KUKA KRL program: makrosps.src

&ACCESS RVO1
&COMMENT MAKRO_SPS_BASIC
&PARAM TEMPLATE = C:\KRC\Roboter\Template\makrospsvorgabe.src
&PARAM TPVW_VERSION = 8.1.8
&PARAM EDITMASK = MakroSPS
DEF MAKROSPS()
   ;FOLD Makro Anfang ;%{PSE}%MKUKATPVW
      SPS_N=-1
   ;ENDFOLD
   ;FOLD -- Freilaufende  SPS  (Basic) -- ;%{E}%MKUKATPVW %CVW_COM %VCOMMENT %P 2:-- Freilaufende  SPS  (Basic) --, 3: VW_COMMENT
   ;ENDFOLD
   ;FOLD -- KS24 -- ;%{E}%MKUKATPVW %CVW_COM %VCOMMENT %P 2:-- KS24 --, 3: VW_COMMENT
   ;ENDFOLD
   ;FOLD -- Version: 01 -- ;%{E}%MKUKATPVW %CVW_COM %VCOMMENT %P 2:-- Version: 01 --, 3: VW_COMMENT
   ;ENDFOLD
   ;FOLD -- Stand: 008 -- ;%{E}%MKUKATPVW %CVW_COM %VCOMMENT %P 2:-- Stand: 008 --, 3: VW_COMMENT
   ;ENDFOLD
   ;FOLD -- letzte  Aenderung  02.11.2017 LZ -- ;%{E}%MKUKATPVW %CVW_COM %VCOMMENT %P 2:-- letzte  Aenderung  02.11.2017 LZ --, 3: VW_COMMENT
   ;ENDFOLD
   ;FOLD -- Hilfszeit MakroSPS -- ;%{E}%MKUKATPVW %CVW_COM %VCOMMENT %P 2:-- Hilfszeit MakroSPS --, 3: VW_COMMENT
   ;ENDFOLD
   ;FOLD t20 ( !A4060 ) = -35[1/10Sek] ;%{E}%MKUKATPVW %CVW_SPS %VTASG %P 2:t20 ( !A4060 ) = -35[1/10Sek], 3: TASG
      VW(#SET_TIME,NOT $OUT[4060],20,0,-35)
   ;ENDFOLD
   ;FOLD -- Hilfsflags fuer Medien -- ;%{E}%MKUKATPVW %CVW_COM %VCOMMENT %P 2:-- Hilfsflags fuer Medien --, 3: VW_COMMENT
   ;ENDFOLD
   ;FOLD F127 = (!F734 & E514 & E515) + (F734 & E517 & E518) ;%{E}%MKUKATPVW %CVW_SPS %VBOASG %P 2:F127 = (!F734 & E514 & E515) + (F734 & E517 & E518), 3: BOASG
      $FLAG[127] = (NOT $FLAG[734] AND $IN[514] AND $IN[515]) OR ($FLAG[734] AND $IN[517] AND $IN[518])
   ;ENDFOLD
   ;FOLD F162 = E522 & E523 ;%{E}%MKUKATPVW %CVW_SPS %VBOASG %P 2:F162 = E522 & E523, 3: BOASG
      $FLAG[162] = $IN[522] AND $IN[523]
   ;ENDFOLD
   ;FOLD F198 = E530 & E531 ;%{E}%MKUKATPVW %CVW_SPS %VBOASG %P 2:F198 = E530 & E531, 3: BOASG
      $FLAG[198] = $IN[530] AND $IN[531]
   ;ENDFOLD
   ;FOLD -- Reset Motorsteuermodul KF 1 -- ;%{E}%MKUKATPVW %CVW_COM %VCOMMENT %P 2:-- Reset Motorsteuermodul KF 1 --, 3: VW_COMMENT
   ;ENDFOLD
   ;FOLD A833 = !T20 & E840 & A4060 + E840 & E26 ;%{E}%MKUKATPVW %CVW_SPS %VBOASG %P 2:A833 = !T20 & E840 & A4060 + E840 & E26, 3: BOASG
      $OUT[833] = NOT $TIMER_FLAG[20] AND $IN[840] AND $OUT[4060] OR $IN[840] AND $IN[26]
   ;ENDFOLD
   ;FOLD -- Reset Motorsteuermodul KS 1 -- ;%{E}%MKUKATPVW %CVW_COM %VCOMMENT %P 2:-- Reset Motorsteuermodul KS 1 --, 3: VW_COMMENT
   ;ENDFOLD
   ;FOLD A841 = !T20 & E848 & A4060 + E848 & E26 ;%{E}%MKUKATPVW %CVW_SPS %VBOASG %P 2:A841 = !T20 & E848 & A4060 + E848 & E26, 3: BOASG
      $OUT[841] = NOT $TIMER_FLAG[20] AND $IN[848] AND $OUT[4060] OR $IN[848] AND $IN[26]
   ;ENDFOLD
   ;FOLD -- Reset Motorsteuermodul ZS 1 -- ;%{E}%MKUKATPVW %CVW_COM %VCOMMENT %P 2:-- Reset Motorsteuermodul ZS 1 --, 3: VW_COMMENT
   ;ENDFOLD
   ;FOLD A849 = !T20 & E856 & A4060 + E856 & E26 ;%{E}%MKUKATPVW %CVW_SPS %VBOASG %P 2:A849 = !T20 & E856 & A4060 + E856 & E26, 3: BOASG
      $OUT[849] = NOT $TIMER_FLAG[20] AND $IN[856] AND $OUT[4060] OR $IN[856] AND $IN[26]
   ;ENDFOLD
   ;FOLD -- Reset Motorsteuermodul KF 2 -- ;%{E}%MKUKATPVW %CVW_COM %VCOMMENT %P 2:-- Reset Motorsteuermodul KF 2 --, 3: VW_COMMENT
   ;ENDFOLD
   ;FOLD A993 = !T20 & E1000 & A4060 + E1000 & E26 ;%{E}%MKUKATPVW %CVW_SPS %VBOASG %P 2:A993 = !T20 & E1000 & A4060 + E1000 & E26, 3: BOASG
      $OUT[993] = NOT $TIMER_FLAG[20] AND $IN[1000] AND $OUT[4060] OR $IN[1000] AND $IN[26]
   ;ENDFOLD
   ;FOLD -- Reset Motorsteuermodul KS 2 -- ;%{E}%MKUKATPVW %CVW_COM %VCOMMENT %P 2:-- Reset Motorsteuermodul KS 2 --, 3: VW_COMMENT
   ;ENDFOLD
   ;FOLD A1001 = !T20 & E1008 & A4060 + E1008 & E26 ;%{E}%MKUKATPVW %CVW_SPS %VBOASG %P 2:A1001 = !T20 & E1008 & A4060 + E1008 & E26, 3: BOASG
      $OUT[1001] = NOT $TIMER_FLAG[20] AND $IN[1008] AND $OUT[4060] OR $IN[1008] AND $IN[26]
   ;ENDFOLD
   ;FOLD -- Reset Motorsteuermodul ZS 2 -- ;%{E}%MKUKATPVW %CVW_COM %VCOMMENT %P 2:-- Reset Motorsteuermodul ZS 2 --, 3: VW_COMMENT
   ;ENDFOLD
   ;FOLD A1009 = !T20 & E1016 & A4060 + E1016 & E26 ;%{E}%MKUKATPVW %CVW_SPS %VBOASG %P 2:A1009 = !T20 & E1016 & A4060 + E1016 & E26, 3: BOASG
      $OUT[1009] = NOT $TIMER_FLAG[20] AND $IN[1016] AND $OUT[4060] OR $IN[1016] AND $IN[26]
   ;ENDFOLD
   ;FOLD -- Reset Motorsteuermodul KF 3 -- ;%{E}%MKUKATPVW %CVW_COM %VCOMMENT %P 2:-- Reset Motorsteuermodul KF 3 --, 3: VW_COMMENT
   ;ENDFOLD
   ;FOLD A1153 = !T20 & E1160 & A4060 + E1160 & E26 ;%{E}%MKUKATPVW %CVW_SPS %VBOASG %P 2:A1153 = !T20 & E1160 & A4060 + E1160 & E26, 3: BOASG
      $OUT[1153] = NOT $TIMER_FLAG[20] AND $IN[1160] AND $OUT[4060] OR $IN[1160] AND $IN[26]
   ;ENDFOLD
   ;FOLD -- Reset Motorsteuermodul KS 3 -- ;%{E}%MKUKATPVW %CVW_COM %VCOMMENT %P 2:-- Reset Motorsteuermodul KS 3 --, 3: VW_COMMENT
   ;ENDFOLD
   ;FOLD A1161 = !T20 & E1168 & A4060 + E1168 & E26 ;%{E}%MKUKATPVW %CVW_SPS %VBOASG %P 2:A1161 = !T20 & E1168 & A4060 + E1168 & E26, 3: BOASG
      $OUT[1161] = NOT $TIMER_FLAG[20] AND $IN[1168] AND $OUT[4060] OR $IN[1168] AND $IN[26]
   ;ENDFOLD
   ;FOLD -- Reset Motorsteuermodul ZS 2 -- ;%{E}%MKUKATPVW %CVW_COM %VCOMMENT %P 2:-- Reset Motorsteuermodul ZS 2 --, 3: VW_COMMENT
   ;ENDFOLD
   ;FOLD A1169 = !T20 & E1176 & A4060 + E1176 & E26 ;%{E}%MKUKATPVW %CVW_SPS %VBOASG %P 2:A1169 = !T20 & E1176 & A4060 + E1176 & E26, 3: BOASG
      $OUT[1169] = NOT $TIMER_FLAG[20] AND $IN[1176] AND $OUT[4060] OR $IN[1176] AND $IN[26]
   ;ENDFOLD
   ;FOLD -- FK von SK1 abspeichern -- ;%{E}%MKUKATPVW %CVW_COM %VCOMMENT %P 2:-- FK von SK1 abspeichern --, 3: VW_COMMENT
   ;ENDFOLD
   ;FOLD F80 = E804 & !E806 & !E775 & E785 + E785 & E15 + F80 & A785 + F525 + E145 ;%{E}%MKUKATPVW %CVW_SPS %VBOASG %P 2:F80 = E804 & !E806 & !E775 & E785 + E785 & E15 + F80 & A785 + F525 + E145, 3: BOASG
      $FLAG[80] = $IN[804] AND NOT $IN[806] AND NOT $IN[775] AND $IN[785] OR $IN[785] AND $IN[15] OR $FLAG[80] AND $OUT[785] OR $FLAG[525] OR $IN[145]
   ;ENDFOLD
   ;FOLD -- FK von Kombi 1 abspeichern -- ;%{E}%MKUKATPVW %CVW_COM %VCOMMENT %P 2:-- FK von Kombi 1 abspeichern --, 3: VW_COMMENT
   ;ENDFOLD
   ;FOLD F833 = E787 & !E789 & !E775 & E719 + E719 & E15 + F833 & A718 + F525 + E130 ;%{E}%MKUKATPVW %CVW_SPS %VBOASG %P 2:F833 = E787 & !E789 & !E775 & E719 + E719 & E15 + F833 & A718 + F525 + E130, 3: BOASG
      $FLAG[833] = $IN[787] AND NOT $IN[789] AND NOT $IN[775] AND $IN[719] OR $IN[719] AND $IN[15] OR $FLAG[833] AND $OUT[718] OR $FLAG[525] OR $IN[130]
   ;ENDFOLD
   ;FOLD -- FK von SK2 abspeichern -- ;%{E}%MKUKATPVW %CVW_COM %VCOMMENT %P 2:-- FK von SK2 abspeichern --, 3: VW_COMMENT
   ;ENDFOLD
   ;FOLD F140 = E964 & !E966 & !E935 & E945 + E945 & E15 + F140 & A945 + F525 + E177 ;%{E}%MKUKATPVW %CVW_SPS %VBOASG %P 2:F140 = E964 & !E966 & !E935 & E945 + E945 & E15 + F140 & A945 + F525 + E177, 3: BOASG
      $FLAG[140] = $IN[964] AND NOT $IN[966] AND NOT $IN[935] AND $IN[945] OR $IN[945] AND $IN[15] OR $FLAG[140] AND $OUT[945] OR $FLAG[525] OR $IN[177]
   ;ENDFOLD
   ;FOLD -- FK von Kombi 2 abspeichern -- ;%{E}%MKUKATPVW %CVW_COM %VCOMMENT %P 2:-- FK von Kombi 2 abspeichern --, 3: VW_COMMENT
   ;ENDFOLD
   ;FOLD F834 = E947 & !E949 & !E935 & E879 + E879 & E15 + F834 & A878 + F525 + E162 ;%{E}%MKUKATPVW %CVW_SPS %VBOASG %P 2:F834 = E947 & !E949 & !E935 & E879 + E879 & E15 + F834 & A878 + F525 + E162, 3: BOASG
      $FLAG[834] = $IN[947] AND NOT $IN[949] AND NOT $IN[935] AND $IN[879] OR $IN[879] AND $IN[15] OR $FLAG[834] AND $OUT[878] OR $FLAG[525] OR $IN[162]
   ;ENDFOLD
   ;FOLD -- FK von SK3 abspeichern -- ;%{E}%MKUKATPVW %CVW_COM %VCOMMENT %P 2:-- FK von SK3 abspeichern --, 3: VW_COMMENT
   ;ENDFOLD
   ;FOLD F176 = E1124 & !E1126 & !E1095 & E1105 + E1105 & E15 + F176 & A1105 + F525 + E209 ;%{E}%MKUKATPVW %CVW_SPS %VBOASG %P 2:F176 = E1124 & !E1126 & !E1095 & E1105 + E1105 & E15 + F176 & A1105 + F525 + E209, 3: BOASG
      $FLAG[176] = $IN[1124] AND NOT $IN[1126] AND NOT $IN[1095] AND $IN[1105] OR $IN[1105] AND $IN[15] OR $FLAG[176] AND $OUT[1105] OR $FLAG[525] OR $IN[209]
   ;ENDFOLD
   ;FOLD -- FK von Kombi 3 abspeichern -- ;%{E}%MKUKATPVW %CVW_COM %VCOMMENT %P 2:-- FK von Kombi 3 abspeichern --, 3: VW_COMMENT
   ;ENDFOLD
   ;FOLD F835 = E1107 & !E1109 & !E1095 & E1039 + E1039 & E15 + F835 & A1038 + F525 + E194 ;%{E}%MKUKATPVW %CVW_SPS %VBOASG %P 2:F835 = E1107 & !E1109 & !E1095 & E1039 + E1039 & E15 + F835 & A1038 + F525 + E194, 3: BOASG
      $FLAG[835] = $IN[1107] AND NOT $IN[1109] AND NOT $IN[1095] AND $IN[1039] OR $IN[1039] AND $IN[15] OR $FLAG[835] AND $OUT[1038] OR $FLAG[525] OR $IN[194]
   ;ENDFOLD
   ;FOLD -- BZ1 -- ;%{E}%MKUKATPVW %CVW_COM %VCOMMENT %P 2:-- BZ1 --, 3: VW_COMMENT
   ;ENDFOLD
   ;FOLD -- A1702 = (!E1697 + !E1699) & E26 -- ;%{E}%MKUKATPVW %CVW_COM %VCOMMENT %P 2:-- A1702 = (!E1697 + !E1699) & E26 --, 3: VW_COMMENT
   ;ENDFOLD
   ;FOLD -- BZ2 -- ;%{E}%MKUKATPVW %CVW_COM %VCOMMENT %P 2:-- BZ2 --, 3: VW_COMMENT
   ;ENDFOLD
   ;FOLD -- A1750 = (!E1745 + !E1747) & E26 -- ;%{E}%MKUKATPVW %CVW_COM %VCOMMENT %P 2:-- A1750 = (!E1745 + !E1747) & E26 --, 3: VW_COMMENT
   ;ENDFOLD
   ;FOLD -- MS1 -- ;%{E}%MKUKATPVW %CVW_COM %VCOMMENT %P 2:-- MS1 --, 3: VW_COMMENT
   ;ENDFOLD
   ;FOLD A1857 = EIN ;%{E}%MKUKATPVW %CVW_SPS %VBOASG %P 2:A1857 = EIN, 3: BOASG
      $OUT[1857] = TRUE
   ;ENDFOLD
   ;FOLD A1858 = !E1858 & (E26 + E27 + !T20 & A4060) ;%{E}%MKUKATPVW %CVW_SPS %VBOASG %P 2:A1858 = !E1858 & (E26 + E27 + !T20 & A4060), 3: BOASG
      $OUT[1858] = NOT $IN[1858] AND ($IN[26] OR $IN[27] OR NOT $TIMER_FLAG[20] AND $OUT[4060])
   ;ENDFOLD
   ;FOLD F570 = A9 & A16 & A4060 & A4039 & E1857 & E1874 & (F960 + F597 & !E128) ;%{E}%MKUKATPVW %CVW_SPS %VBOASG %P 2:F570 = A9 & A16 & A4060 & A4039 & E1857 & E1874 & (F960 + F597 & !E128), 3: BOASG
      $FLAG[570] = $OUT[9] AND $OUT[16] AND $OUT[4060] AND $OUT[4039] AND $IN[1857] AND $IN[1874] AND ($FLAG[960] OR $FLAG[597] AND NOT $IN[128])
   ;ENDFOLD
   ;FOLD A1859 = A12 & E12 & F570 & F571 & (E1859 + !E26) + E211 & F570 & F571 ;%{E}%MKUKATPVW %CVW_SPS %VBOASG %P 2:A1859 = A12 & E12 & F570 & F571 & (E1859 + !E26) + E211 & F570 & F571, 3: BOASG
      $OUT[1859] = $OUT[12] AND $IN[12] AND $FLAG[570] AND $FLAG[571] AND ($IN[1859] OR NOT $IN[26]) OR $IN[211] AND $FLAG[570] AND $FLAG[571]
   ;ENDFOLD
   ;FOLD -- MS2 -- ;%{E}%MKUKATPVW %CVW_COM %VCOMMENT %P 2:-- MS2 --, 3: VW_COMMENT
   ;ENDFOLD
   ;FOLD A1889 = EIN ;%{E}%MKUKATPVW %CVW_SPS %VBOASG %P 2:A1889 = EIN, 3: BOASG
      $OUT[1889] = TRUE
   ;ENDFOLD
   ;FOLD A1890 = !E1890 & (E26 + E27 + !T20 & A4060) ;%{E}%MKUKATPVW %CVW_SPS %VBOASG %P 2:A1890 = !E1890 & (E26 + E27 + !T20 & A4060), 3: BOASG
      $OUT[1890] = NOT $IN[1890] AND ($IN[26] OR $IN[27] OR NOT $TIMER_FLAG[20] AND $OUT[4060])
   ;ENDFOLD
   ;FOLD F579 = A9 & A16 & A4060 & A4039 & E1889 & E1906 & (F960 + F597 & !E128) ;%{E}%MKUKATPVW %CVW_SPS %VBOASG %P 2:F579 = A9 & A16 & A4060 & A4039 & E1889 & E1906 & (F960 + F597 & !E128), 3: BOASG
      $FLAG[579] = $OUT[9] AND $OUT[16] AND $OUT[4060] AND $OUT[4039] AND $IN[1889] AND $IN[1906] AND ($FLAG[960] OR $FLAG[597] AND NOT $IN[128])
   ;ENDFOLD
   ;FOLD A1891 = A12 & E12 & F579 & F580 & (E1891 + !E26) + E203 & F579 & F580 ;%{E}%MKUKATPVW %CVW_SPS %VBOASG %P 2:A1891 = A12 & E12 & F579 & F580 & (E1891 + !E26) + E203 & F579 & F580, 3: BOASG
      $OUT[1891] = $OUT[12] AND $IN[12] AND $FLAG[579] AND $FLAG[580] AND ($IN[1891] OR NOT $IN[26]) OR $IN[203] AND $FLAG[579] AND $FLAG[580]
   ;ENDFOLD
   ;FOLD -- KL1 -- ;%{E}%MKUKATPVW %CVW_COM %VCOMMENT %P 2:-- KL1 --, 3: VW_COMMENT
   ;ENDFOLD
   ;FOLD A1527 = A10 + E1568 ;%{E}%MKUKATPVW %CVW_SPS %VBOASG %P 2:A1527 = A10 + E1568, 3: BOASG
      $OUT[1527] = $OUT[10] OR $IN[1568]
   ;ENDFOLD
   ;FOLD A1528 = A12 ;%{E}%MKUKATPVW %CVW_SPS %VBOASG %P 2:A1528 = A12, 3: BOASG
      $OUT[1528] = $OUT[12]
   ;ENDFOLD
   ;FOLD F339 = (A1529 + A1535 + E9 & !E15 & !F336) & !E1551 & A10 ;%{E}%MKUKATPVW %CVW_SPS %VBOASG %P 2:F339 = (A1529 + A1535 + E9 & !E15 & !F336) & !E1551 & A10, 3: BOASG
      $FLAG[339] = ($OUT[1529] OR $OUT[1535] OR $IN[9] AND NOT $IN[15] AND NOT $FLAG[336]) AND NOT $IN[1551] AND $OUT[10]
   ;ENDFOLD
   ;FOLD A1547 = (F339 & !T20 + F337 + E168) & F542 ;%{E}%MKUKATPVW %CVW_SPS %VBOASG %P 2:A1547 = (F339 & !T20 + F337 + E168) & F542, 3: BOASG
      $OUT[1547] = ($FLAG[339] AND NOT $TIMER_FLAG[20] OR $FLAG[337] OR $IN[168]) AND $FLAG[542]
   ;ENDFOLD
   ;FOLD A1550 = (F339 & !T20 + F337 + E168) & F542 & !E15 ;%{E}%MKUKATPVW %CVW_SPS %VBOASG %P 2:A1550 = (F339 & !T20 + F337 + E168) & F542 & !E15, 3: BOASG
      $OUT[1550] = ($FLAG[339] AND NOT $TIMER_FLAG[20] OR $FLAG[337] OR $IN[168]) AND $FLAG[542] AND NOT $IN[15]
   ;ENDFOLD
   ;FOLD -- KL2 -- ;%{E}%MKUKATPVW %CVW_COM %VCOMMENT %P 2:-- KL2 --, 3: VW_COMMENT
   ;ENDFOLD
   ;FOLD A1591 = A10 + E1632 ;%{E}%MKUKATPVW %CVW_SPS %VBOASG %P 2:A1591 = A10 + E1632, 3: BOASG
      $OUT[1591] = $OUT[10] OR $IN[1632]
   ;ENDFOLD
   ;FOLD A1592 = A12 ;%{E}%MKUKATPVW %CVW_SPS %VBOASG %P 2:A1592 = A12, 3: BOASG
      $OUT[1592] = $OUT[12]
   ;ENDFOLD
   ;FOLD F360 = (A1593 + A1599 + E9 & !E15 & !F357) & !E1615 & A10 ;%{E}%MKUKATPVW %CVW_SPS %VBOASG %P 2:F360 = (A1593 + A1599 + E9 & !E15 & !F357) & !E1615 & A10, 3: BOASG
      $FLAG[360] = ($OUT[1593] OR $OUT[1599] OR $IN[9] AND NOT $IN[15] AND NOT $FLAG[357]) AND NOT $IN[1615] AND $OUT[10]
   ;ENDFOLD
   ;FOLD A1611 = (F360 & !T20 + F358 + E184) & F543 ;%{E}%MKUKATPVW %CVW_SPS %VBOASG %P 2:A1611 = (F360 & !T20 + F358 + E184) & F543, 3: BOASG
      $OUT[1611] = ($FLAG[360] AND NOT $TIMER_FLAG[20] OR $FLAG[358] OR $IN[184]) AND $FLAG[543]
   ;ENDFOLD
   ;FOLD A1614 = (F360 & !T20 + F358 + E184) & F543 & !E15 ;%{E}%MKUKATPVW %CVW_SPS %VBOASG %P 2:A1614 = (F360 & !T20 + F358 + E184) & F543 & !E15, 3: BOASG
      $OUT[1614] = ($FLAG[360] AND NOT $TIMER_FLAG[20] OR $FLAG[358] OR $IN[184]) AND $FLAG[543] AND NOT $IN[15]
   ;ENDFOLD
   ;FOLD -- KL3 -- ;%{E}%MKUKATPVW %CVW_COM %VCOMMENT %P 2:-- KL3 --, 3: VW_COMMENT
   ;ENDFOLD
   ;FOLD A1655 = A10 + E1696 ;%{E}%MKUKATPVW %CVW_SPS %VBOASG %P 2:A1655 = A10 + E1696, 3: BOASG
      $OUT[1655] = $OUT[10] OR $IN[1696]
   ;ENDFOLD
   ;FOLD A1656 = A12 ;%{E}%MKUKATPVW %CVW_SPS %VBOASG %P 2:A1656 = A12, 3: BOASG
      $OUT[1656] = $OUT[12]
   ;ENDFOLD
   ;FOLD F381 = (A1657 + A1663 + E9 & !E15 & !F378) & !E1679 & A10 ;%{E}%MKUKATPVW %CVW_SPS %VBOASG %P 2:F381 = (A1657 + A1663 + E9 & !E15 & !F378) & !E1679 & A10, 3: BOASG
      $FLAG[381] = ($OUT[1657] OR $OUT[1663] OR $IN[9] AND NOT $IN[15] AND NOT $FLAG[378]) AND NOT $IN[1679] AND $OUT[10]
   ;ENDFOLD
   ;FOLD A1675 = (F381 & !T20 + F379 + E200) & F544 ;%{E}%MKUKATPVW %CVW_SPS %VBOASG %P 2:A1675 = (F381 & !T20 + F379 + E200) & F544, 3: BOASG
      $OUT[1675] = ($FLAG[381] AND NOT $TIMER_FLAG[20] OR $FLAG[379] OR $IN[200]) AND $FLAG[544]
   ;ENDFOLD
   ;FOLD A1678 = (F381 & !T20 + F379 + E200) & F544 & !E15 ;%{E}%MKUKATPVW %CVW_SPS %VBOASG %P 2:A1678 = (F381 & !T20 + F379 + E200) & F544 & !E15, 3: BOASG
      $OUT[1678] = ($FLAG[381] AND NOT $TIMER_FLAG[20] OR $FLAG[379] OR $IN[200]) AND $FLAG[544] AND NOT $IN[15]
   ;ENDFOLD
   ;FOLD -- CZ1 Servo / CZ1 Pneum. -- ;%{E}%MKUKATPVW %CVW_COM %VCOMMENT %P 2:-- CZ1 Servo / CZ1 Pneum. --, 3: VW_COMMENT
   ;ENDFOLD
   ;FOLD A1345 = (E26 + E27 + F489) & (E1424 & F538 & !F539 + !F538 & F539 & E1368) ;%{E}%MKUKATPVW %CVW_SPS %VBOASG %P 2:A1345 = (E26 + E27 + F489) & (E1424 & F538 & !F539 + !F538 & F539 & E1368), 3: BOASG
      $OUT[1345] = ($IN[26] OR $IN[27] OR $FLAG[489]) AND ($IN[1424] AND $FLAG[538] AND NOT $FLAG[539] OR NOT $FLAG[538] AND $FLAG[539] AND $IN[1368])
   ;ENDFOLD
   ;FOLD -- CZ2 Servo / CZ2 Pneum. -- ;%{E}%MKUKATPVW %CVW_COM %VCOMMENT %P 2:-- CZ2 Servo / CZ2 Pneum. --, 3: VW_COMMENT
   ;ENDFOLD
   ;FOLD A1425 = (E26 + E27 + F489) & (E1504 & F540 & !F541 + !F540 & F541 & E1448) ;%{E}%MKUKATPVW %CVW_SPS %VBOASG %P 2:A1425 = (E26 + E27 + F489) & (E1504 & F540 & !F541 + !F540 & F541 & E1448), 3: BOASG
      $OUT[1425] = ($IN[26] OR $IN[27] OR $FLAG[489]) AND ($IN[1504] AND $FLAG[540] AND NOT $FLAG[541] OR NOT $FLAG[540] AND $FLAG[541] AND $IN[1448])
   ;ENDFOLD
   ;FOLD -- NZ1 Servo / NZ1 Hydr. -- ;%{E}%MKUKATPVW %CVW_COM %VCOMMENT %P 2:-- NZ1 Servo / NZ1 Hydr. --, 3: VW_COMMENT
   ;ENDFOLD
   ;FOLD A1185 = (E26 + E27 + F489) & (E1264 & F534 & !F535 + F534 & !F535 & E1216) ;%{E}%MKUKATPVW %CVW_SPS %VBOASG %P 2:A1185 = (E26 + E27 + F489) & (E1264 & F534 & !F535 + F534 & !F535 & E1216), 3: BOASG
      $OUT[1185] = ($IN[26] OR $IN[27] OR $FLAG[489]) AND ($IN[1264] AND $FLAG[534] AND NOT $FLAG[535] OR $FLAG[534] AND NOT $FLAG[535] AND $IN[1216])
   ;ENDFOLD
   ;FOLD -- NZ2 Servo / NZ2 Hydr. -- ;%{E}%MKUKATPVW %CVW_COM %VCOMMENT %P 2:-- NZ2 Servo / NZ2 Hydr. --, 3: VW_COMMENT
   ;ENDFOLD
   ;FOLD A1265 = (E26 + E27 + F489) & (E1344 & F536 & !F537 + !F536 & F537 & E1296) ;%{E}%MKUKATPVW %CVW_SPS %VBOASG %P 2:A1265 = (E26 + E27 + F489) & (E1344 & F536 & !F537 + !F536 & F537 & E1296), 3: BOASG
      $OUT[1265] = ($IN[26] OR $IN[27] OR $FLAG[489]) AND ($IN[1344] AND $FLAG[536] AND NOT $FLAG[537] OR NOT $FLAG[536] AND $FLAG[537] AND $IN[1296])
   ;ENDFOLD
   ;FOLD -- RW1 -- ;%{E}%MKUKATPVW %CVW_COM %VCOMMENT %P 2:-- RW1 --, 3: VW_COMMENT
   ;ENDFOLD
   ;FOLD A1265 = (E26 + E27 + F489) & E1328 & F479 & F478 ;%{E}%MKUKATPVW %CVW_SPS %VBOASG %P 2:A1265 = (E26 + E27 + F489) & E1328 & F479 & F478, 3: BOASG
      $OUT[1265] = ($IN[26] OR $IN[27] OR $FLAG[489]) AND $IN[1328] AND $FLAG[479] AND $FLAG[478]
   ;ENDFOLD
   ;FOLD -- RW2 -- ;%{E}%MKUKATPVW %CVW_COM %VCOMMENT %P 2:-- RW2 --, 3: VW_COMMENT
   ;ENDFOLD
   ;FOLD A1185 = (E26 + E27 + F489) & E1248 & F484 & F483 ;%{E}%MKUKATPVW %CVW_SPS %VBOASG %P 2:A1185 = (E26 + E27 + F489) & E1248 & F484 & F483, 3: BOASG
      $OUT[1185] = ($IN[26] OR $IN[27] OR $FLAG[489]) AND $IN[1248] AND $FLAG[484] AND $FLAG[483]
   ;ENDFOLD
   ;FOLD -- Ohne Prozess in Single Step -- ;%{E}%MKUKATPVW %CVW_COM %VCOMMENT %P 2:-- Ohne Prozess in Single Step --, 3: VW_COMMENT
   ;ENDFOLD
   ;FOLD F525 = F525 & A11 ;%{E}%MKUKATPVW %CVW_SPS %VBOASG %P 2:F525 = F525 & A11, 3: BOASG
      $FLAG[525] = $FLAG[525] AND $OUT[11]
   ;ENDFOLD
   ;FOLD -- Roboter in Single Step -- ;%{E}%MKUKATPVW %CVW_COM %VCOMMENT %P 2:-- Roboter in Single Step --, 3: VW_COMMENT
   ;ENDFOLD
   ;FOLD F985 = A11 ;%{E}%MKUKATPVW %CVW_SPS %VBOASG %P 2:F985 = A11, 3: BOASG
      $FLAG[985] = $OUT[11]
   ;ENDFOLD
   ;FOLD -- Online Freigabe Roboter -- ;%{E}%MKUKATPVW %CVW_COM %VCOMMENT %P 2:-- Online Freigabe Roboter --, 3: VW_COMMENT
   ;ENDFOLD
   ;FOLD A127 = M128 ;%{E}%MKUKATPVW %CVW_SPS %VBOASG %P 2:A127 = M128, 3: BOASG
      $OUT[127] = $CYCFLAG[128]
   ;ENDFOLD
   ;FOLD A128 = M129 ;%{E}%MKUKATPVW %CVW_SPS %VBOASG %P 2:A128 = M129, 3: BOASG
      $OUT[128] = $CYCFLAG[129]
   ;ENDFOLD
   ; FOLD ;%{H}
END
; ENDFOLD
